VAR_GLOBAL PERSISTENT
	
/////////////////////////////////////////////////////////////////////////////////////Log/////////////////////////////////////////////////////////////////////////////////////
	
	stUserLog					: ARRAY [0..250] OF ST_UserLog;
	
	aDataHistory				: ARRAY[0..200] OF ST_CycleData;
	astEventsHistory			: ARRAY[0..200] OF ST_EventsHistory;
	stJavasCriptPDF				: ST_JavasCriptPDF;

	stProbesSettings			: ST_ProbesSettings;

END_VAR

(* stored: Version 1.1.0.1, ProductVersion 3.1.4026.17
   GVL GVL_Persistent: Id {c4d03ea6-35af-4633-972d-fef3cfe7daa9} *)
